KUKA KRL data list: calc_block_placement.dat

&ACCESS RV1
DEFDAT  calc_block_placement PUBLIC

ENDDAT
